INTERFACE I_Component
VAR_INPUT
	sName			: STRING[20];
	bEnable     	: BOOL;
	bStart      	: BOOL;
	bHalt			: BOOL;
	bStop       	: BOOL;
	eMode       	: E_ComponentMode; 		// 0=OFF, 1=AUTO, 2=MANUAL
END_VAR

VAR_OUTPUT
	eState			: E_ComponentState;		// 0=READY, 1=BUSY, 2=DONE
	iErrorCode		: INT;
	sStatusText 	: STRING[50];
END_VAR

METHOD Halt : BOOL
VAR_INPUT
END_VAR
END_METHOD

METHOD Start : BOOL
VAR_INPUT
END_VAR
END_METHOD

METHOD Stop : BOOL
VAR_INPUT
END_VAR
END_METHOD

END_INTERFACE

(* stored: Version 1.1.0.1, ProductVersion 3.1.4024.15
   Itf I_Component: Id {3337d348-193e-4804-bc6d-8f5b2d280baf}
   Method Halt: Id {65f0acb6-737d-487e-a1b7-0fd6741c7d88}
   Method Start: Id {d12c8e5a-4245-4c17-b9b0-a0ee94e9265a}
   Method Stop: Id {4d9a5b11-9982-4955-97b8-a30e468e1c2f} *)
